// Renishaw BiSS-C absolute encoder used with an EL5042
TYPE ST_RenishawAbsEnc :
STRUCT
    Count AT %I*: ULINT; // Connect to encoder "Position" input
    Status: ST_EL5042_Status; // Status struct placeholder
    Ref: ULINT; // Encoder zero position (useful for aligned position with gantries)
END_STRUCT
END_TYPE

(* stored: Version 1.1.0.1
   DUT ST_RenishawAbsEnc: Id {6f5997cc-f148-4e63-9185-dfba8067f4f0} *)
